FUNCTION_BLOCK Station001_Components EXTENDS TcoCore.TcoObject
VAR	
	{attribute addProperty Name "Horizontal cyclinder A1"}
	_horizontal : fbPiston(THIS^);
	{attribute addProperty Name "Vertical cyclinder A2"}
	_vertical : fbPiston(THIS^);
	{attribute addProperty Name "Gripper A3"}
	_gripper : fbPiston(THIS^);	

	{attribute addProperty Name "Digital input"}
	_di : TcoDi(THIS^);	
	{attribute addProperty Name "Wrapped component example 1"}
	_wrappedComponent1 : Example1WrappedComponent(THIS^);	
	
	{attribute addProperty Name "Wrapped component example 2"}
	_wrappedComponent2 : Example2WrappedComponent(THIS^);	
	
	{attribute clr [RenderIgnore()]}
	_wrappedComponents: Example2WrappedComponents;
	tempSisgnal: BOOL;
	temp2Sisgnal: BOOL;
END_VAR

VAR
	_simTimerValue : UINT := 500;
	_simTimer : Tc2_Standard.TON;
END_VAR

_vertical();
_vertical.Service();
_horizontal();
_gripper();

_wrappedComponent1();


_wrappedComponent2.Components.digitalInput(inoSignal:=tempSisgnal);
_wrappedComponent2.Components.digitaOutput(inoSignal:=temp2Sisgnal);

_wrappedComponent2();

_simTimer(IN := TRUE, PT := UINT_TO_TIME(_simTimerValue));
SimulateCylinder(_vertical);
SimulateCylinder(_horizontal);
SimulateCylinder(_gripper);

PROPERTY Gripper : IPistonGripper
GET
Gripper := _gripper;
END_GET
END_PROPERTY

PROPERTY Horizontal : IPistonHorizontal
GET
Horizontal := _horizontal;
END_GET
END_PROPERTY

METHOD SimulateCylinder
VAR_IN_OUT
	ioCyclinder : fbPiston;
END_VAR
ioCyclinder.iHomePositionSensor := ioCyclinder.qHomePositionActuator AND _simTimer.Q;
ioCyclinder.iWorkPositionSensor := ioCyclinder.qWorkPositionActuator AND _simTimer.Q;
END_METHOD

PROPERTY Vertical : IPistonVertical
GET
Vertical := _vertical;
END_GET
END_PROPERTY

END_FUNCTION_BLOCK

(* stored: Version 1.1.0.1
   POU Station001_Components: Id {973f80ae-5d0f-02e7-24c7-363a147de04a}, SpecialFunc None
   Property Gripper: Id {6a01dc28-d982-0fb5-2745-9e809c451913}
   Get Get: Id {610a8cd9-7ae4-08af-1bc0-99ccfbc7becf}
   Property Horizontal: Id {92e43ad3-5c26-0dec-2c49-d1ed9b4a55ad}
   Get Get: Id {024846ec-1132-0b00-2fcf-2b664b0d337e}
   Method SimulateCylinder: Id {b1ee2641-008c-0760-1502-d9d6bdf50ae0}
   Property Vertical: Id {ebb87fc4-eb98-0125-1c02-13275d3bc4b7}
   Get Get: Id {a74c9db1-1590-07ad-1319-bdaa0e2438bf} *)
